// TIA Portal V18 export
ORGANIZATION_BLOCK "Main"   // OB1, FBD, ProgramCycle
TITLE = "Main Program Sweep (Cycle)"
{ S7_Optimized_Access := 'TRUE' }
VERSION : 0.1
// stored: AutoNumber true, IsIECCheckEnabled false, SetENOAutomatically false
   VAR_INPUT
      Initial_Call : Bool;   // Initial call of this OB
      Remanence : Bool;   // =True, if remanent data are available
   END_VAR
   VAR_TEMP
      Diag_Ret_Value1 : Int;
   END_VAR
BEGIN

REGION Network 1: Module State of a PROFINET Dev
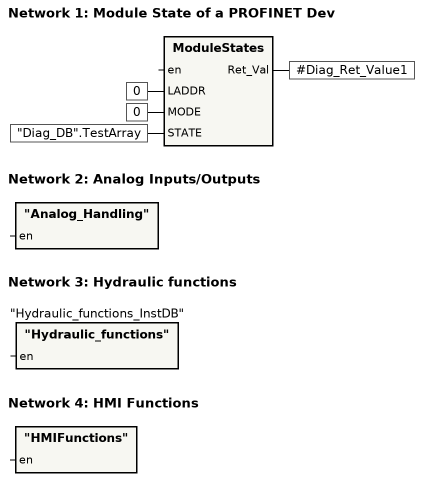
   #Diag_Ret_Value1 := ModuleStates(LADDR := 0, MODE := 0, STATE := "Diag_DB".TestArray);
END_REGION

REGION Network 2: Analog Inputs/Outputs
   "Analog_Handling"();
END_REGION

REGION Network 3: Hydraulic functions
   "Hydraulic_functions_InstDB"();   // "Hydraulic_functions"
END_REGION

REGION Network 4: HMI Functions
   "HMIFunctions"();
END_REGION
END_ORGANIZATION_BLOCK
